{attribute 'GeneratedUsingTerminal: EP3744-0041-0016'}
{attribute addProperty BoxType "EP3744-0041-0016"}
{attribute addProperty Id "StatusAT %I*Status_F2CE6D917ValueAT %I*DINT4"}
{attribute addProperty CRC "1159803140"}
{attribute addProperty Size "11"}
TYPE AI_Inputs_Channel_45213104 EXTENDS InputBase_8311D824 :
STRUCT
	{attribute addProperty Name "Status"}
	Status AT %I* : Status_F2CE6D91;
	{attribute addProperty Name "Value"}
	Value AT %I* : DINT;
END_STRUCT
END_TYPE

(* stored: Version 1.2.0.0, ProductVersion 3.1.4024.11
   DUT AI_Inputs_Channel_45213104: Id {14738129-fd36-442f-9506-9b35f26e59e3} *)
